_CFC_ (* Continuous Function Chart, elements in execution order *)
#0 TON_sost_VKL:TON(IN: SHU6_P2_UST_SOST_VKL, PT: T#500ms)
#1 RT_VKL:R_TRIG(CLK: #0.Q)
#2 AND(#1.Q, NOT SHU6_P2_UST_RE_PROGREV)
#3 FT_PROGREV:F_TRIG(CLK: SHU6_P2_UST_RE_PROGREV)
#4 OR(#2, #3.Q)
#5 OR(SHU6_P2_UST_SOST_OTKL, SHU6_P2_B45)
#6 RS_Pusk:RS(SET: #4, RESET1: #5)
#7 SHU6_P2_UST_RE_PUSK <= #6.Q1
_END_CFC_
(* the same logic as Structured Text *)
TON_sost_VKL(IN := SHU6_P2_UST_SOST_VKL, PT := T#500ms);
RT_VKL(CLK := TON_sost_VKL.Q);
FT_PROGREV(CLK := SHU6_P2_UST_RE_PROGREV);
RS_Pusk(SET := (RT_VKL.Q AND NOT SHU6_P2_UST_RE_PROGREV) OR FT_PROGREV.Q, RESET1 := SHU6_P2_UST_SOST_OTKL OR SHU6_P2_B45);
SHU6_P2_UST_RE_PUSK := RS_Pusk.Q1;
END_PROGRAM

(* POU Regim/Rabota, CFC *)
PROGRAM Rabota
VAR
	RS_Rabota: RS;
	FT_Pusk: F_TRIG;
END_VAR
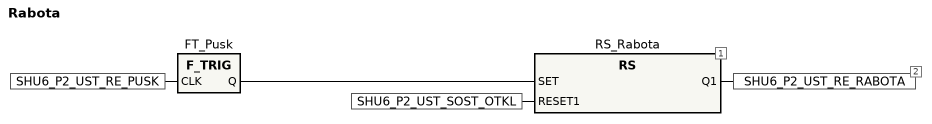
_CFC_ (* Continuous Function Chart, elements in execution order *)
#0 FT_Pusk:F_TRIG(CLK: SHU6_P2_UST_RE_PUSK)
#1 RS_Rabota:RS(SET: #0.Q, RESET1: SHU6_P2_UST_SOST_OTKL)
#2 SHU6_P2_UST_RE_RABOTA <= #1.Q1
_END_CFC_
(* the same logic as Structured Text *)
FT_Pusk(CLK := SHU6_P2_UST_RE_PUSK);
RS_Rabota(SET := FT_Pusk.Q, RESET1 := SHU6_P2_UST_SOST_OTKL);
SHU6_P2_UST_RE_RABOTA := RS_Rabota.Q1;
END_PROGRAM

(* POU IM/ALL_IM, CFC *)
PROGRAM ALL_IM
VAR
END_VAR
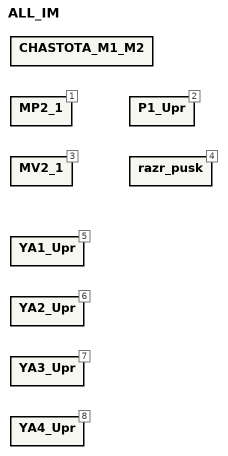
_CFC_ (* Continuous Function Chart, elements in execution order *)
#0 CHASTOTA_M1_M2()
#1 MP2_1()
#2 P1_Upr()
#3 MV2_1()
#4 razr_pusk()
#5 YA1_Upr()
#6 YA2_Upr()
#7 YA3_Upr()
#8 YA4_Upr()
_END_CFC_
(* the same logic as Structured Text *)
CHASTOTA_M1_M2();
MP2_1();
P1_Upr();
MV2_1();
razr_pusk();
YA1_Upr();
YA2_Upr();
YA3_Upr();
YA4_Upr();
END_PROGRAM

(* POU IM/MP2/CHASTOTA_M1_M2, CFC *)
PROGRAM CHASTOTA_M1_M2
VAR
	RR: RAMP_REAL;
	SR_START_STER_REG: SR;
	SR_START_POV_REG: RS;
	RT_KOMVKL: R_TRIG;
	RT_KOMVKL_2: R_TRIG;
	RT_KOMVKL_1: R_TRIG;
	Zad_PE: TON;
	RS_RUCH: RS;
	V_RUCH: BOOL;
	TON_RUCH: TON;
	SHU6_P2_M_MAXSPEED_CH_OLD: REAL;
	TON_STER_1: TON;
	TON_STER_2: TON;
	RT_PDK: R_TRIG;
	FT_PDK: F_TRIG;
END_VAR
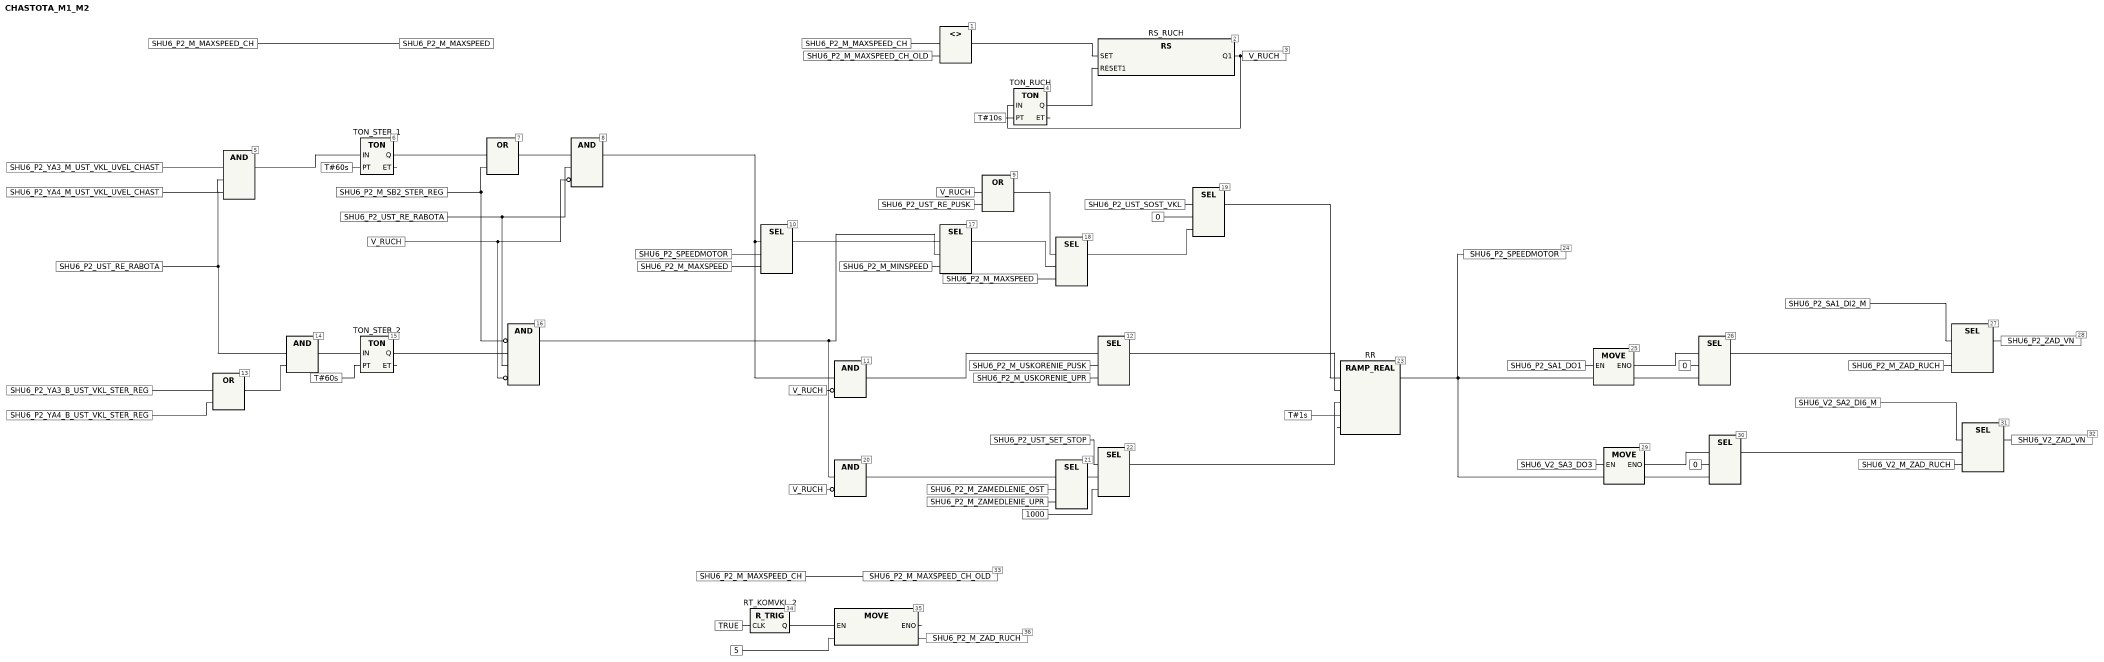
